FUNCTION_BLOCK SuperBohrmachine IMPLEMENTS I_SuperBohrmachine
VAR_INPUT
END_VAR
VAR_OUTPUT
END_VAR
VAR
	fbBohrkopf: Bohrkopf;
	fbAxesManager: AxesManager;
	stConfig: ST_Config;
	
	eZustand: E_STATES_SUPERBOHRMACHINE := E_STATES_SUPERBOHRMACHINE.stopped;
	
	// Stop-Command set via outside call?
	bDoStop: BOOL := FALSE;
	
	// anzufahrende Punkte
	aPunkte: ARRAY [0..3] OF ST_2DPoint;
	nCurIdx: USINT := 0;
END_VAR

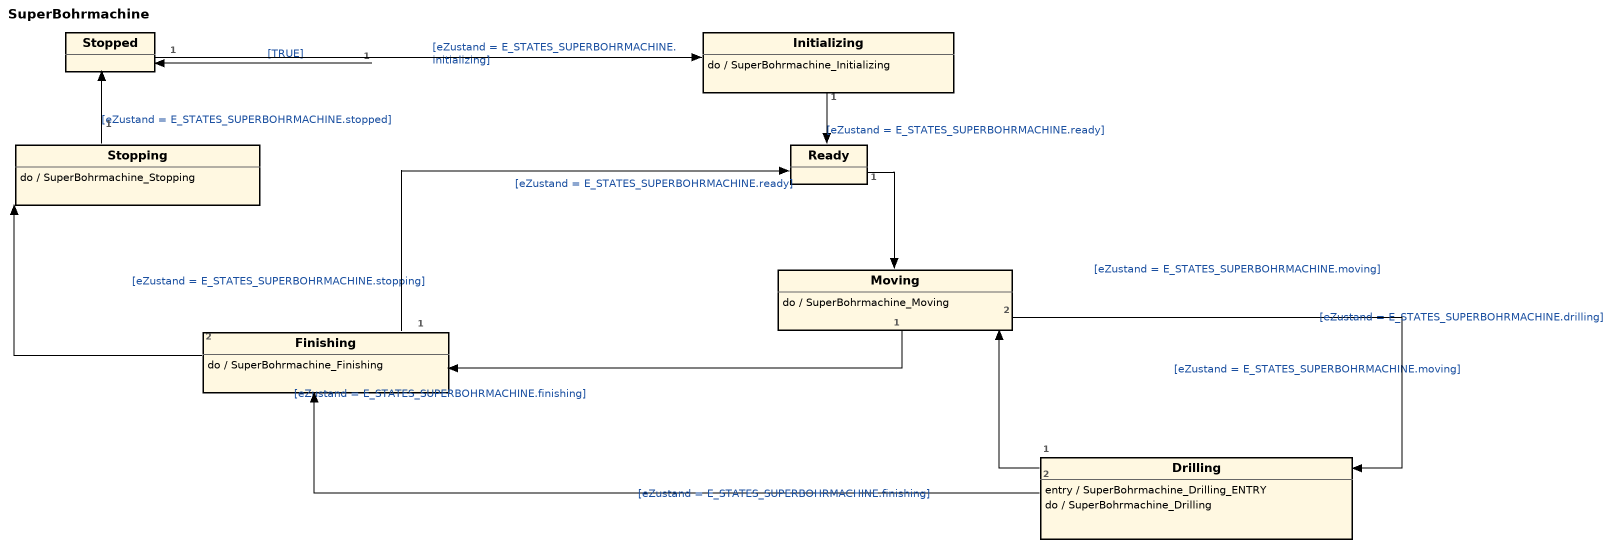
STATECHART SuperBohrmachine  // abortable
    START StartState1
    STATE Stopped
    STATE Initializing
        do / SuperBohrmachine_Initializing
    STATE Stopping
        do / SuperBohrmachine_Stopping
    STATE Ready
    STATE Moving
        do / SuperBohrmachine_Moving
    STATE Finishing
        do / SuperBohrmachine_Finishing
    STATE Drilling
        entry / SuperBohrmachine_Drilling_ENTRY
        do / SuperBohrmachine_Drilling
    StartState1 -> Stopped [TRUE] // priority 1, on completion
    Stopped -> Initializing [eZustand = E_STATES_SUPERBOHRMACHINE.initializing] // priority 1
    Initializing -> Ready [eZustand = E_STATES_SUPERBOHRMACHINE.ready] // priority 1
    Stopping -> Stopped [eZustand = E_STATES_SUPERBOHRMACHINE.stopped] // priority 1
    Ready -> Moving [eZustand = E_STATES_SUPERBOHRMACHINE.moving] // priority 1
    Moving -> Finishing [eZustand = E_STATES_SUPERBOHRMACHINE.finishing] // priority 1
    Moving -> Drilling [eZustand = E_STATES_SUPERBOHRMACHINE.drilling] // priority 2
    Finishing -> Ready [eZustand = E_STATES_SUPERBOHRMACHINE.ready] // priority 1
    Finishing -> Stopping [eZustand = E_STATES_SUPERBOHRMACHINE.stopping] // priority 2
    Drilling -> Moving [eZustand = E_STATES_SUPERBOHRMACHINE.moving] // priority 1
    Drilling -> Finishing [eZustand = E_STATES_SUPERBOHRMACHINE.finishing] // priority 2
END_STATECHART

METHOD Bohren : HRESULT
CASE eZustand OF
	E_STATES_SUPERBOHRMACHINE.ready:
		THIS^.eZustand := E_STATES_SUPERBOHRMACHINE.moving;
		Bohren := S_OK;
		
	ELSE
		Bohren := S_FALSE;

END_CASE
END_METHOD

PROPERTY PUBLIC Config : ST_Config
SET
VAR
	rBreite: LREAL;
	rLaenge: LREAL;
	rAbstand: LREAL := 10;
END_VAR
stConfig := Config;

// Punkte berechnen
rBreite := stConfig.rBreite;
rLaenge := stConfig.rLaenge;

// Punkt 1
aPunkte[0].x := rAbstand;
aPunkte[0].y := rAbstand;

// Punkt 2
aPunkte[1].x := 10;
aPunkte[1].y := rBreite - rAbstand;

// Punkt 3
aPunkte[2].x := rLaenge - rAbstand;
aPunkte[2].y := rBreite - rAbstand;

// Punkt 4
aPunkte[3].x := rLaenge - rAbstand;
aPunkte[3].y := rAbstand;

fbBohrkopf.Config REF= stConfig;
END_SET
END_PROPERTY

METHOD Start : HRESULT
VAR_INPUT
	config: REFERENCE TO ST_Config;
END_VAR
CASE eZustand OF
	E_STATES_SUPERBOHRMACHINE.stopped:
		// Konfiguration setzen
		THIS^.Config := config;
		// Anlage starten
		THIS^.eZustand := E_STATES_SUPERBOHRMACHINE.initializing;
		Start := S_PENDING;
		
	E_STATES_SUPERBOHRMACHINE.ready:
		Start := S_OK;
		
	ELSE
		Start := S_PENDING;
	
END_CASE
END_METHOD

METHOD Stop : HRESULT
CASE eZustand OF
	// Anlage gestoppt
	E_STATES_SUPERBOHRMACHINE.stopped:
		Stop := S_OK;
	
	E_STATES_SUPERBOHRMACHINE.finishing:
		// Stop während normalem Finishing
		THIS^.bDoStop := TRUE;
		Stop := S_PENDING;

	E_STATES_SUPERBOHRMACHINE.stopping:
		Stop := S_PENDING;

	ELSE
		// Anlage stoppen
		THIS^.bDoStop := TRUE;
		THIS^.eZustand := E_STATES_SUPERBOHRMACHINE.finishing;
		
END_CASE
END_METHOD

METHOD PRIVATE SuperBohrmachine_Drilling : BOOL
VAR_INPUT
END_VAR

IF fbBohrkopf.Ready THEN
	// fertig gebohrt
	eZustand := E_STATES_SUPERBOHRMACHINE.moving;
END_IF
END_METHOD

METHOD PRIVATE SuperBohrmachine_Drilling_ENTRY : BOOL
VAR_INPUT
END_VAR
fbBohrkopf.Bohren();
END_METHOD

METHOD PRIVATE SuperBohrmachine_Finishing : BOOL
VAR
	stHomePoint: ST_2DPoint := (x := 0, y := 0);
END_VAR
VAR_INST
	bAxesHomeDone: BOOL := FALSE;
	bBohrkopfUpDone: BOOL := FALSE;
END_VAR
(*
1. Bohrkopf hochfahren
2. AxesManager zum Nullpunkt fahren
3. bDoStop = TRUE ? 'stopping' : 'ready'
*)

fbBohrkopf.GoUp(Done => bBohrkopfUpDone);

IF bBohrkopfUpDone THEN
	fbAxesManager.GoTo(stHomePoint, Done => bAxesHomeDone);
	IF bAxesHomeDone THEN
		bAxesHomeDone := FALSE;
		bBohrkopfUpDone := FALSE;
		// Anlage stoppen oder Bearbeitung fertig?
		IF bDoStop THEN
			eZustand := E_STATES_SUPERBOHRMACHINE.stopping;
		ELSE
			eZustand := E_STATES_SUPERBOHRMACHINE.ready;
		END_IF
	END_IF
END_IF
END_METHOD

METHOD PRIVATE SuperBohrmachine_Initializing : BOOL
VAR_INPUT
END_VAR
(*
- AxesManager initialisieren
- Bohrkopf initialisieren
*)

fbAxesManager.Init();
fbBohrkopf.Init();

IF fbAxesManager.Initialized AND fbBohrkopf.Initialized THEN
	// Anlage initialisiert
	eZustand := E_STATES_SUPERBOHRMACHINE.ready;
END_IF
END_METHOD

METHOD PRIVATE SuperBohrmachine_Moving : BOOL
VAR_INPUT
END_VAR
IF nCurIdx = 4 THEN
	// letzter Punkt wurde gebohrt => State 'finishing'
	nCurIdx := 0;
	eZustand := E_STATES_SUPERBOHRMACHINE.finishing;
ELSE
	// Zum Punkt fahren => State 'drilling'
	IF fbAxesManager.GoTo(aPunkte[nCurIdx]) THEN
		nCurIdx := nCurIdx + 1;
		eZustand := E_STATES_SUPERBOHRMACHINE.drilling;
	END_IF
END_IF
END_METHOD

METHOD PRIVATE SuperBohrmachine_Stopping : BOOL
VAR CONSTANT
	stHomePoint: ST_2DPoint := (x := 0, y := 0);
END_VAR
VAR_INST
	bAxesStopDone: BOOL := FALSE;
	bBohrkopfStopDone: BOOL := FALSE;
END_VAR
(*
- Bohrkopf-Achsen stoppen
- AxesManager stop
*)

fbBohrkopf.Stop();
fbAxesManager.Stop();


IF fbAxesManager.Stopped AND fbBohrkopf.Stopped THEN
	bDoStop := FALSE;
	eZustand := E_STATES_SUPERBOHRMACHINE.stopped;
END_IF
END_METHOD

END_FUNCTION_BLOCK

(* stored: Version 1.1.0.1, ProductVersion 3.1.4024.3
   POU SuperBohrmachine: Id {3a09d3d9-90b0-4be2-a068-25b1a8ba9f03}, SpecialFunc None
   Method Bohren: Id {4297fade-6109-4cd6-92ea-76b00fe2b146}
   Property Config: Id {8db9cb02-e528-41a3-9750-6cdc189f145c}
   Set Set: Id {2b5d076e-8edc-459d-b597-84d378a7e41f}
   Method Start: Id {693e534a-741d-4d7e-92df-75d91daa7887}
   Method Stop: Id {98892f86-fd9a-4b22-a1a4-f9c700833f2d}
   Method SuperBohrmachine_Drilling: Id {053a03e9-9512-4bcd-a2f7-9ce5ee8bf34e}
   Method SuperBohrmachine_Drilling_ENTRY: Id {f7b81aca-b880-416b-829d-f7369b60f714}
   Method SuperBohrmachine_Finishing: Id {e72c143e-d393-4ffc-b695-602d0a72cb5e}
   Method SuperBohrmachine_Initializing: Id {a18a4640-ed5f-4513-b1db-e2c0d6eef25d}
   Method SuperBohrmachine_Moving: Id {905066dc-2bd7-480c-ab68-d90733d8c277}
   Method SuperBohrmachine_Stopping: Id {1f7c71f8-35f7-452d-9946-a6cdf4595e57} *)
